FUNCTION_BLOCK L1_stul_FBD
VAR_INPUT
	CO1: BOOL;
	C5DPR: BOOL;
	C4DPR: BOOL;
END_VAR
VAR_OUTPUT
	MO: BOOL;
	M5DPR: BOOL;
	M4DPR: BOOL;
END_VAR
VAR
END_VAR

// NETWORK 1

END_FUNCTION_BLOCK

(* stored: Version 1.1.0.1, ProductVersion 3.1.4024.13
   POU L1_stul_FBD: Id {5b2e8084-ae15-493a-822c-6e5f23ddf242}, SpecialFunc None *)
